FUNCTION_BLOCK FeedPumpFlowSp (* Basic Function Block Type *)
  (* Standard: 61499-2 *)
  (* Version 0.0, 7/3/2024, SESA713705, Schneider Electric, Template *)
  PACKAGE SE.Nereda;
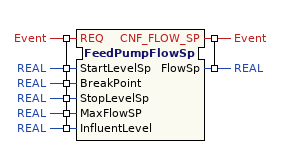
  EVENT_INPUT
    REQ WITH InfluentLevel, StartLevelSp, BreakPoint, StopLevelSp, MaxFlowSP;
  END_EVENT
  EVENT_OUTPUT
    CNF_FLOW_SP WITH FlowSp;
  END_EVENT
  VAR_INPUT
    StartLevelSp : REAL;
    BreakPoint : REAL;
    StopLevelSp : REAL;
    MaxFlowSP : REAL;
    InfluentLevel : REAL;
  END_VAR
  VAR_OUTPUT
    FlowSp : REAL;
  END_VAR
  VAR
    a : REAL;
    b : REAL;
  END_VAR
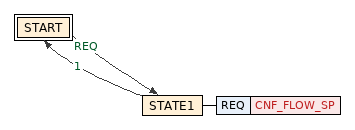
  EC_STATES
    START; (* Initial State *)
    STATE1 : REQ -> CNF_FLOW_SP;
  END_STATES
  EC_TRANSITIONS
    START TO STATE1 := REQ;
    STATE1 TO START := 1;
  END_TRANSITIONS
  ALGORITHM REQ IN ST: (* Normally executed algorithm *)
;
IF InfluentLevel < StartLevelSp OR InfluentLevel < BreakPoint THEN
		FlowSp := MaxFlowSP;

ELSIF BreakPoint <= InfluentLevel AND InfluentLevel <= StopLevelSp THEN
	a := MaxFlowSP / (BreakPoint - StopLevelSp);
	b := MaxFlowSP * StopLevelSp / (StopLevelSp - BreakPoint);
	FlowSp := a * InfluentLevel +b;

ELSE
	FlowSp := 0;
END_IF;
  END_ALGORITHM
END_FUNCTION_BLOCK
